# EPICS autosave request: current/autosave/thermocon.req
# iocAdmin autosave template
# Format:
# <PVNAME>
$(IOC):ACCESS
$(IOC):CA_CLNT_CNT.HIGH
$(IOC):CA_CLNT_CNT.HIHI
$(IOC):CA_CONN_CNT.HIGH
$(IOC):CA_CONN_CNT.HIHI
$(IOC):SUSP_TASK_CNT.HIHI
$(IOC):FD_FREE.LOW
$(IOC):FD_FREE.LOLO
$(IOC):IOC_CPU_LOAD.HIGH
$(IOC):IOC_CPU_LOAD.HIHI
$(IOC):MEM_FREE.LOW
$(IOC):MEM_FREE.LOLO
$(IOC):START_CNT
$(IOC):MEM_BLK_FREE.LOW
$(IOC):MEM_BLK_FREE.LOLO
$(BASE):CTRL_OP_SET
$(BASE):TARG_TEMP_SET
